TYPE ST_InfoDataGroup :
STRUCT
	usiMapState:USINT;
	usiMapDiag:USINT;
END_STRUCT
END_TYPE

(* stored: Version 1.1.0.1, ProductVersion 3.1.0.20
   DUT ST_InfoDataGroup: Id {ae06926f-e8bf-4119-b822-5528fb116efe} *)
